(* PLC project One Station VGP, Blank VGP 1.0 *)
(* stored: creationDateTime 2016-05-18T21:14:07, modificationDateTime 2020-03-25T22:35:50 *)

PROGRAM My_Program
  VAR
    Level AT %IW0 : INT;
    min_sp AT %QW1 : INT;
    max_sp AT %QW2 : INT;
    mode_register AT %QW3 : INT;
    pump_register AT %QW4 : INT;
    valve_register AT %QW5 : INT;
    pump AT %QX0.0 : BOOL;
    valve AT %QX0.1 : BOOL;
  END_VAR
  VAR  (* added by the conversion: wires and edge detectors of the diagram *)
    _EQ44_ENO : BOOL;
    _EQ44_OUT : BOOL;
    _EQ7_OUT : BOOL;
    _EQ11_ENO : BOOL;
    _EQ11_OUT : BOOL;
    _GE93_ENO : BOOL;
    _GE93_OUT : BOOL;
  END_VAR

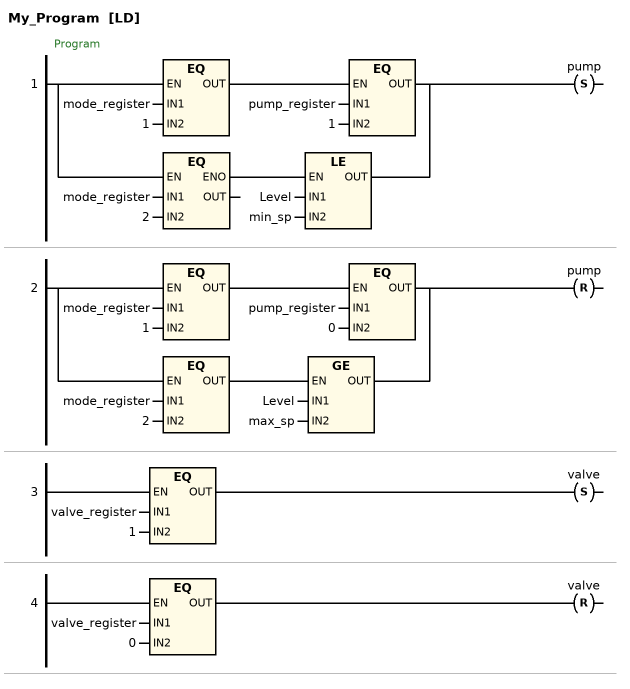
(* LD diagram, written out as Structured Text *)
(* Program *)
_EQ44_OUT := EQ(EN := mode_register = 1, IN1 := pump_register, IN2 := 1, ENO => _EQ44_ENO);
_EQ7_OUT := mode_register = 2;
IF _EQ44_OUT OR Level <= min_sp THEN pump := TRUE; END_IF;
_EQ11_OUT := EQ(EN := mode_register = 1, IN1 := pump_register, IN2 := 0, ENO => _EQ11_ENO);
_GE93_OUT := GE(EN := mode_register = 2, IN1 := Level, IN2 := max_sp, ENO => _GE93_ENO);
IF _EQ11_OUT OR _GE93_OUT THEN pump := FALSE; END_IF;
IF valve_register = 1 THEN valve := TRUE; END_IF;
IF valve_register = 0 THEN valve := FALSE; END_IF;
END_PROGRAM

CONFIGURATION Config0
  RESOURCE Res0 ON PLC
    TASK TaskMain(INTERVAL := T#50ms, PRIORITY := 0);
    PROGRAM Inst0 WITH TaskMain : My_Program;
  END_RESOURCE
END_CONFIGURATION
